FUNCTION ADC_10V : REAL
VAR_INPUT
	normal_input : REAL;
	x_max : REAL := 10;
	x_min : REAL := 0;
END_VAR
VAR
	voltage_reading : REAL;
END_VAR

// 0 - 10V AI INPUT | normal_input 0-100%
voltage_reading := 10 * normal_input;
ADC_10V := (voltage_reading - x_min) / (x_max - x_min);

END_FUNCTION

(* stored: Version 1.1.0.1, ProductVersion 3.1.4024.11
   POU ADC_10V: Id {2a4913c1-96ae-4091-b40a-f5f7b5005c01}, SpecialFunc None *)
